FUNCTION_BLOCK PUBLIC FB_IO
VAR_INPUT
	PTTT: REFERENCE TO ARRAY [1.. GVL_IO.cNumofPT] OF FB_PressureTransducer;
END_VAR
VAR
	inlet:FB_matrix;
	fill:FB_matrix;
	dispense:FB_matrix;
	nsensorNumber:INT;
	rows:INT;
	cols:INT;
	aInletMAtrixValveCmds: INT;
END_VAR

M_PTTTransducers();
M_Solenoids();

PROPERTY DispenseMatrix : FB_matrix
SET
dispense := DispenseMatrix;
END_SET
END_PROPERTY

PROPERTY FillMatrix : FB_matrix
SET
fill := FillMatrix;
END_SET
END_PROPERTY

PROPERTY InletMatrix : FB_matrix
SET
inlet := InletMatrix;
END_SET
END_PROPERTY

METHOD M_PTTTransducers
FOR nsensorNumber:=1 TO GVL_IO.cNumofPT DO		
    PTTT[nsensorNumber].RawPressure := GVL_IO.aPressRaw[nsensorNumber];
    PTTT[nsensorNumber].RawTemperature := GVL_IO.aTempRaw[nsensorNumber];
END_FOR
END_METHOD

METHOD M_Solenoids
//Update IO for valve commands
FOR rows:=1 TO GVL_HMI.cInletRows DO
	FOR cols:=1 TO GVL_HMI.cInletCols DO
	    GVL_IO.aInletMAtrixValveCmds[rows,cols]:= inlet.aValveCommands[rows,cols];
	END_FOR
END_FOR
FOR rows:=1 TO GVL_HMI.cMaxRows DO
	FOR cols:=1 TO GVL_HMI.cMaxCols DO
	    GVL_IO.aFillMatrixValveCmds[rows,cols]:= fill.aValveCommands[rows,cols];
		GVL_IO.aDispenseMatrixValveCmds[rows,cols]:= Dispense.aValveCommands[rows,cols];
	END_FOR
END_FOR
END_METHOD

END_FUNCTION_BLOCK

(* stored: Version 1.1.0.1
   POU FB_IO: Id {1c9b80c2-f6a7-4a98-9c0f-22ba5373f0a7}, SpecialFunc None
   Folder Actuators: Id {0a74f44c-a186-4f5d-abba-c1f92f894549}
   Folder Properties: Id {1bea0c20-9e15-4457-b2ac-582c67937e90}
   Folder Sensors: Id {2415513d-42f8-4814-955f-fcef3eafc61a}
   Property DispenseMatrix: Id {25f8c8ea-72db-4e7f-9424-df95763ea36e}
   Set Set: Id {b4b61de5-0f59-4900-bd91-af2c73760bee}
   Property FillMatrix: Id {eb86371d-b4e3-4663-8fa9-8f44d0dcee82}
   Set Set: Id {76f52427-6cad-4e42-b8f0-ed73ad49d5b8}
   Property InletMatrix: Id {19664f95-51b4-4ed3-a2b7-b542e5c6a464}
   Set Set: Id {17f0b4eb-6d50-4ab9-a197-cba0365312ee}
   Method M_PTTTransducers: Id {db9ee37e-2b9d-4ae2-ba7d-052f24f151f3}
   Method M_Solenoids: Id {dbd95f87-3564-46ed-86ee-3bfcb091fedb} *)
